// TwinCAT 3 PLC project A_SimpleLogMessage
// ProgramVersion: 3.1.4023.0
// libraries:
//   Log4TC, * (mbc engineering GmbH)
//   Tc2_Standard, * (Beckhoff Automation GmbH)
//   Tc2_System, * (Beckhoff Automation GmbH)
//   Tc3_Module, * (Beckhoff Automation GmbH)
// project tree:
//   / MAIN.TcPOU, PlcTask.TcTTO
// (motion and I/O tree: see PLC project loggingexample)
// real-time tasks:
//   TASK PlcTask: cycle T#10ms, priority 20, ADS port 350
//   TASK PlcTask1: cycle T#10ms, priority 21, ADS port 351
//   TASK PlcTask2: cycle T#10ms, priority 22, ADS port 352

CONFIGURATION A_SimpleLogMessage
    RESOURCE PLC ON TwinCAT3
        TASK PlcTask(INTERVAL := T#10ms, PRIORITY := 20);
        PROGRAM MAIN WITH PlcTask : MAIN;
    END_RESOURCE
END_CONFIGURATION

// ---- MAIN.TcPOU
PROGRAM MAIN

IF _TaskInfo[GETCURTASKINDEXEX()].FirstCycle THEN
	F_Log(E_LogLevel.eInfo, 'SPS Task gestartet.');
END_IF

PRG_TaskLog.Call();

END_PROGRAM
